TYPE ReadXmlProcessArgs :
STRUCT
	///Full path of the filename to read
	filePath: STRING;
END_STRUCT
END_TYPE

(* stored: Version 1.1.0.1, ProductVersion 3.1.4019.2
   DUT ReadXmlProcessArgs: Id {2d3a400e-6a57-4643-80fd-f4fd13142988} *)
